// TIA Portal V17 program export: 1 tag tables, 4 data types, 4 data blocks, 9 code blocks (in call order from the OBs), 0 instance data blocks

VAR_GLOBAL   // PLC tag table "Default tag table"
   M1_out AT %Q200.0 : "M_out";
   M1_in AT %I200.0 : "M_in";
   M2_out AT %Q219.0 : "M_out";
   M2_in AT %I209.0 : "M_in";
   M3_out AT %Q238.0 : "M_out";
   M3_in AT %I218.0 : "M_in";
   M4_out AT %Q257.0 : "M_out";
   M4_in AT %I227.0 : "M_in";
   M5_out AT %Q276.0 : "M_out";
   M5_in AT %I236.0 : "M_in";
   M6_out AT %Q295.0 : "M_out";
   M6_in AT %I245.0 : "M_in";
   M7_out AT %Q314.0 : "M_out";
   M7_in AT %I254.0 : "M_in";
   M8_out AT %Q333.0 : "M_out";
   M8_in AT %I263.0 : "M_in";
   M9_out AT %Q352.0 : "M_out";
   M9_in AT %I272.0 : "M_in";
   M10_out AT %Q371.0 : "M_out";
   M10_in AT %I281.0 : "M_in";
   M11_out AT %Q390.0 : "M_out";
   M11_in AT %I290.0 : "M_in";
   M12_out AT %Q409.0 : "M_out";
   M12_in AT %I299.0 : "M_in";
   M13_out AT %Q428.0 : "M_out";
   M13_in AT %I308.0 : "M_in";
   M14_out AT %Q447.0 : "M_out";
   M14_in AT %I317.0 : "M_in";
   M15_out AT %Q466.0 : "M_out";
   M15_in AT %I326.0 : "M_in";
   M16_out AT %Q485.0 : "M_out";
   M16_in AT %I335.0 : "M_in";
   M17_out AT %Q504.0 : "M_out";
   M17_in AT %I344.0 : "M_in";
   M18_out AT %Q523.0 : "M_out";
   M18_in AT %I353.0 : "M_in";
END_VAR

TYPE "M_in"
VERSION : 0.1
   STRUCT
      statusword : "M_in_status_w";
      act_speed { S7_SetPoint := 'True'} : DInt;   // Velocity Actual Value - 606Ch
      last_alarm { S7_SetPoint := 'True'} : UInt;   // Error Code - 603Fh
      curr_mode_operation { ExternalAccessible := 'False'; ExternalVisible := 'False'; ExternalWritable := 'False'} : Byte;   // Modes Of Operation Display - 6061h
   END_STRUCT;

END_TYPE

TYPE "M_in_status_w"
VERSION : 0.1
   STRUCT
      bit_0 : Bool;   // Ready to Switch On
      bit_1 : Bool;   // Switch On
      bit_2 : Bool;   // Operation Enabled
      bit_3 : Bool;   // Fault
      bit_4 : Bool;   // Voltage Enabled
      bit_5 : Bool;   // Quick Stop
      bit_6 : Bool;   // Switch On Disable
      bit_7 : Bool;   // Warning (not used in Axor’s drives)
      bit_8 : Bool;   // Manufacturer specific (not used in Axor’s drives)
      bit_9 : Bool;   // Remote (not used in Axor’s drives)
      bit_10 : Bool;   // Target Reached
      bit_11 : Bool;   // Internal Limit Active
      bit_12 : Bool;   // Speed (standstill)
      bit_13 : Bool;   // Max sleep error (not used in Axor’s drives)
      bit_14 : Bool;   // Manufacturer specific (not used in Axor’s drives)
      bit_15 : Bool;   // Manufacturer specific (not used in Axor’s drives)
   END_STRUCT;

END_TYPE

TYPE "M_out"
VERSION : 0.1
   STRUCT
      controlword { S7_SetPoint := 'False'} : "M_out_control_w";
      sp_speed { S7_SetPoint := 'True'} : DInt;   // Target Velocity - 60FFh
      sp_acc { S7_SetPoint := 'True'} : UDInt;   // Profile Acceleration - 6083h
      sp_dec { S7_SetPoint := 'True'} : UDInt;   // Profile Deceleration - 6084h
      sp_q_stop { S7_SetPoint := 'True'} : UDInt;   // Quick Stop Deceleration - 6085h
      set_mode_op { ExternalAccessible := 'False'; ExternalVisible := 'False'; ExternalWritable := 'False'} : Byte;   // Modes Of Operation - 6060h
   END_STRUCT;

END_TYPE

TYPE "M_out_control_w"
VERSION : 0.1
   STRUCT
      bit_0 { ExternalAccessible := 'False'; ExternalVisible := 'False'; ExternalWritable := 'False'} : Bool;   // Switch On
      bit_1 { ExternalAccessible := 'False'; ExternalVisible := 'False'; ExternalWritable := 'False'} : Bool;   // Enable Voltage
      bit_2 { ExternalAccessible := 'False'; ExternalVisible := 'False'; ExternalWritable := 'False'} : Bool;   // Quick Stop
      bit_3 { ExternalAccessible := 'False'; ExternalVisible := 'False'; ExternalWritable := 'False'} : Bool;   // Operation Enable
      bit_4 { ExternalAccessible := 'False'; ExternalVisible := 'False'; ExternalWritable := 'False'} : Bool;   // Reserved (not used in Axor’s drives)
      bit_5 { ExternalAccessible := 'False'; ExternalVisible := 'False'; ExternalWritable := 'False'} : Bool;   // Reserved (not used in Axor’s drives)
      bit_6 { ExternalAccessible := 'False'; ExternalVisible := 'False'; ExternalWritable := 'False'} : Bool;   // Reserved (not used in Axor’s drives)
      bit_7 { ExternalAccessible := 'False'; ExternalVisible := 'False'; ExternalWritable := 'False'} : Bool;   // Fault Reset
      bit_8 { ExternalAccessible := 'False'; ExternalVisible := 'False'; ExternalWritable := 'False'} : Bool;   // Halt
      bit_9 { ExternalAccessible := 'False'; ExternalVisible := 'False'; ExternalWritable := 'False'} : Bool;   // Reserved (not used in Axor’s drives)
      bit_10 { ExternalAccessible := 'False'; ExternalVisible := 'False'; ExternalWritable := 'False'} : Bool;   // Reserved (not used in Axor’s drives)
      bit_11 { ExternalAccessible := 'False'; ExternalVisible := 'False'; ExternalWritable := 'False'} : Bool;   //  Manufacturer specific (not used in Axor’s drives)
      bit_12 { ExternalAccessible := 'False'; ExternalVisible := 'False'; ExternalWritable := 'False'} : Bool;   //  Manufacturer specific (not used in Axor’s drives)
      bit_13 { ExternalAccessible := 'False'; ExternalVisible := 'False'; ExternalWritable := 'False'} : Bool;   //  Manufacturer specific (not used in Axor’s drives)
      bit_14 { ExternalAccessible := 'False'; ExternalVisible := 'False'; ExternalWritable := 'False'} : Bool;   //  Manufacturer specific (not used in Axor’s drives)
      bit_15 { ExternalAccessible := 'False'; ExternalVisible := 'False'; ExternalWritable := 'False'} : Bool;   //  Manufacturer specific (not used in Axor’s drives)
   END_STRUCT;

END_TYPE

DATA_BLOCK "Main_Safety_RTG1_DB"
{ DB_Accessible_From_OPC_UA := 'FALSE' ;
 S7_Optimized_Access := 'TRUE' }
NAME : FUSI
VERSION : 0.1
NON_RETAIN
"Main_Safety_RTG1"

BEGIN

END_DATA_BLOCK

DATA_BLOCK "instance_ciclo_mac"
{ DB_Accessible_From_OPC_UA := 'FALSE' ;
 S7_Optimized_Access := 'TRUE' }
AUTHOR : Frj
VERSION : 0.1
NON_RETAIN
"ciclo_macchina"

BEGIN

END_DATA_BLOCK

DATA_BLOCK "M1_datiCiclo_DB"
{ DB_Accessible_From_OPC_UA := 'FALSE' ;
 S7_Optimized_Access := 'TRUE' }
VERSION : 0.1
NON_RETAIN
   VAR 
      M1_startProfilo { ExternalAccessible := 'False'; ExternalVisible := 'False'; ExternalWritable := 'False'} : Bool;
      M1_SP_Velocity { ExternalAccessible := 'False'; ExternalVisible := 'False'; ExternalWritable := 'False'} : DInt;
      M1_SP_Acc { ExternalAccessible := 'False'; ExternalVisible := 'False'; ExternalWritable := 'False'} : UDInt;
      M1_SP_Dec { ExternalAccessible := 'False'; ExternalVisible := 'False'; ExternalWritable := 'False'} : UDInt;
      M1_F { ExternalAccessible := 'False'; ExternalVisible := 'False'; ExternalWritable := 'False'} : Int;   // measurement distance for one revolution of the driving shaft of the gearbox [Um]
      M1_SP_QuickStop { ExternalAccessible := 'False'; ExternalVisible := 'False'; ExternalWritable := 'False'} : UDInt;
   END_VAR


BEGIN

END_DATA_BLOCK

DATA_BLOCK "M1_instance_DB"
{ DB_Accessible_From_OPC_UA := 'FALSE' ;
 S7_Optimized_Access := 'TRUE' }
AUTHOR : Frj
VERSION : 0.1
NON_RETAIN
"device_control"

BEGIN
   M_out.set_mode_op := 16#03;

END_DATA_BLOCK

ORGANIZATION_BLOCK "Main"   // OB1, LAD, ProgramCycle
TITLE = "Main Program Sweep (Cycle)"
{ S7_Optimized_Access := 'TRUE' }
VERSION : 0.1
// stored: AutoNumber true, IsIECCheckEnabled false, SetENOAutomatically false
   VAR_INPUT
      Initial_Call : Bool;   // Initial call of this OB
      Remanence : Bool;   // =True, if remanent data are available
   END_VAR
BEGIN

REGION Network 1 (SCL): test velocità lettura dati
   // "M1_out".sp_speed := "M1_out".sp_speed + 1;
   // IF "M1_out".sp_speed > 10000 THEN
   //     "M1_out".sp_speed := 0;
   // END_IF;

   // "M1_out".sp_acc := "M1_out".sp_acc + 1;
   // IF "M1_out".sp_acc > 10000 THEN
   //     "M1_out".sp_acc := 0;
   // END_IF;
END_REGION

REGION Network 2 (SCL): Motore 1
   "M1_instance_DB"(M_in := "M1_in",
                    M_out => "M1_out");


   "instance_ciclo_mac"();
END_REGION
END_ORGANIZATION_BLOCK

FUNCTION_BLOCK "device_control"
TITLE = axor
{ S7_Optimized_Access := 'TRUE' }
AUTHOR : Frj
VERSION : 0.1
   VAR 
      step { ExternalAccessible := 'False'; ExternalVisible := 'False'; ExternalWritable := 'False'} : Int;
   END_VAR

   VAR CONSTANT 
      start : Int := 0;
      not_ready_to_switch_on : Int := 1;
      switch_on_disable : Int := 2;
      ready_to_switch_on : Int := 3;
      switch_on : Int := 4;
      operation_enable : Int := 5;
      quick_stop_active : Int := 6;
      fault : Int := 7;
   END_VAR


BEGIN
	
	
	
	
	
	
	CASE #step OF
	    #start:  // Statement section case 1
	        ;
	    #not_ready_to_switch_on:  // Statement section case 2 to 4
	        ;
	    #switch_on_disable:  // Statement section case 1
	        ;
	    #ready_to_switch_on:  // Statement section case 2 to 4
	        ;
	    #switch_on:  // Statement section case 1
	        ;
	    #operation_enable:  // Statement section case 2 to 4
	        ;
	    #quick_stop_active:  // Statement section case 1
	        ;
	    #fault:  // Statement section case 2 to 4
	        ;
	END_CASE;
	
	
	
END_FUNCTION_BLOCK

FUNCTION_BLOCK "ciclo_macchina"
TITLE = axor
{ S7_Optimized_Access := 'TRUE' }
AUTHOR : Frj
VERSION : 0.1

BEGIN
	REGION Profilo ciclico
	    
	    
	END_REGION
	
	
	
	
	
	
	REGION M1_parametri
	    "M1_instance_DB".startMotor := "M1_datiCiclo_DB".M1_startProfilo;
	    "M1_instance_DB".M_out.set_mode_op := 3; //Profile Velocity
	    
	    "M1_instance_DB".M_out.sp_speed := ("M1_datiCiclo_DB".M1_SP_Velocity * 65536) / "M1_datiCiclo_DB".M1_F;
	    "M1_instance_DB".M_out.sp_acc := ("M1_datiCiclo_DB".M1_SP_Acc * 65536) / "M1_datiCiclo_DB".M1_F;
	    "M1_instance_DB".M_out.sp_dec := ("M1_datiCiclo_DB".M1_SP_Dec * 65536) / "M1_datiCiclo_DB".M1_F;
	    "M1_instance_DB".M_out.sp_q_stop := ("M1_datiCiclo_DB".M1_SP_QuickStop * 65536) / "M1_datiCiclo_DB".M1_F;
	    
	    
	END_REGION
	
	
	
	
	
	
	
	
END_FUNCTION_BLOCK

FUNCTION_BLOCK "LADblock"   // FB7, LAD
{ S7_Optimized_Access := 'TRUE' }
VERSION : 0.1
// stored: AutoNumber true, IsIECCheckEnabled false, IsRetainMemResEnabled false, MemoryReserve 100, SetENOAutomatically false, UDAEnableTagReadback false
BEGIN
END_FUNCTION_BLOCK

FUNCTION_BLOCK "Main_Safety_RTG1"   // FB1, F_FBD
{ S7_Optimized_Access := 'TRUE' }
VERSION : 0.1
// stored: AutoNumber false, IsIECCheckEnabled false, UDAEnableTagReadback false
BEGIN
END_FUNCTION_BLOCK

FUNCTION_BLOCK "STLblock"   // FB6, STL
{ S7_Optimized_Access := 'TRUE' }
VERSION : 0.1
// stored: AutoNumber true, IsRetainMemResEnabled false, MemoryReserve 100, UDAEnableTagReadback false
   VAR
      "int" { ExternalAccessible := 'False'; ExternalVisible := 'False'; ExternalWritable := 'False'} : Int;
   END_VAR
BEGIN

NETWORK
TITLE = 
      L     100;
      T     #"int";


END_FUNCTION_BLOCK

FUNCTION_BLOCK "device_status"
TITLE = axor
{ S7_Optimized_Access := 'TRUE' }
AUTHOR : Frj
VERSION : 0.1
   VAR 
      step { ExternalAccessible := 'False'; ExternalVisible := 'False'; ExternalWritable := 'False'} : Int;
   END_VAR

   VAR CONSTANT 
      start : Int := 0;
      not_ready_to_switch_on : Int := 1;
      switch_on_disable : Int := 2;
      ready_to_switch_on : Int := 3;
      switch_on : Int := 4;
      error : Int := 5;
      spare : Int := 100;
   END_VAR


BEGIN
	
	
	
	
	
	
	CASE #step OF
	    #start:  // Statement section case 1
	        ;
	    #not_ready_to_switch_on:  // Statement section case 2 to 4
	        ;
	    #switch_on_disable:  // Statement section case 1
	        ;
	    #ready_to_switch_on:  // Statement section case 2 to 4
	        ;
	    #switch_on:  // Statement section case 1
	        ;
	        #error:
	            ;
	       
	        
	END_CASE;
	
	
	
END_FUNCTION_BLOCK

FUNCTION_BLOCK "gitFB"
{ S7_Optimized_Access := 'TRUE' }
VERSION : 0.1

BEGIN
END_FUNCTION_BLOCK

FUNCTION_BLOCK "newFB"
{ S7_Optimized_Access := 'TRUE' }
VERSION : 0.1
   VAR 
      iVar { ExternalAccessible := 'False'; ExternalVisible := 'False'; ExternalWritable := 'False'} : Int;
   END_VAR


BEGIN
	#iVar := 2;
	
	#iVar := #iVar;
	
	
END_FUNCTION_BLOCK
